(* Schneider Machine Expert - Basic project demo3, file version 2.2.0.0 *)
(* CompanyInformations: WebSite=https://ics-cybersecurity.academy *)
(* ProjectInformations: Name=ICSJWG demo 3 and +, Description=Demonstrate how to program the PLC so that the SCADA can collect some interesting data for cybersecurity *)
(* UserInformations: LastName=Arnaud, FirstName=SOULLIE, Email=asoullie@ics-cybersecurity.academy *)

HARDWARE
  Cpu 0: TM221ME16R/G
  EthernetConfiguration: NetworkName=M221, IpAllocationMode=FixedAddress, IpAddress=192.168.0.53, SubnetMask=255.255.255.0
  SerialLineConfiguration: Baud=Baud19200, Parity=ParityEven, DataBits=DataBits8, StopBits=StopBits1, PhysicalMedium=PhysicalMediumRs485, TransmissionMode=TransmissionModeModbusRtu, SlaveId=1, Addressing=SlaveAddressing
  MastTask: UsePeriodScanMode=false, PeriodScan=100
  FastTask: Period=255
  CpuBehavior: StartingMode=StartAsPreviousState, AutoSaveRamOnEeprom=true, WatchdogPeriod=250

SYMBOLS  (address, symbol, comment, settings)
  %M0       TIMER_START
  %M20      WASH_INTAKE
  %M23      BARREL_VALVE
  %M100     IO_FORCED
  %M101     INPUT_FORCED
  %M102     OUTPUT_FORCED
  %S12      SB_RUNMODE  "The controller is running"
  %S14      SB_IOFORCED  "This bit indicates there is at least one input or output forced"
  %S15      SB_INFORCED  "This bit indicates there is at least one input forced"
  %S16      SB_OUTFORCED  "This bit indicates there is at least one output forced"
  %SW6      SW_CONTROLSTATUS  "Controller Status: NO CONFIG (0), STOP (2), RUN (3), HALT (4), POWERLESS MODE (5)"
  %SW7      SW_STATE  "This word shows the state of the controller (see online help for details)"
  %SW15     SW_FW1VERSION  "Contains the Firmware version of the controller (1st word)"
  %SW16     SW_FW2VERSION  "Contains the Firmware version of the controller (2nd word)"
  %SW30     SW_LASTSCAN1  "Shows execution time of the last controller scan cycle (in ms).If the scan time is 2,250 ms, %SW30 = 2 and %SW70 = 250"
  %SW70     SW_LASTSCAN2  "Shows the microseconds of the execution time of the last controller scan cycle. If the scan time is 2,250 ms the %SW30 will be 2 and the %SW70 = 250"
  %SW94     SW_SIGNATURE  "Contains the signature, changes in case of an application change, in terms of configuration or programming data"
  %MW0      TIMER_DURATION
  %MW10     STILL_TEMP
  %MW11     STILL_LEVEL
  %MW12     CONDENSER_TEMP
  %MW13     BARREL_LEVEL
  %MW21     HEATER
  %MW22     COOLING_PUMP
  %MW100    BOOTLOADER_VERSION
  %MW101    COMMERCIAL_VERSION
  %MW102    FIRMWARE_V_PART1
  %MW103    FIRMWARE_V_PART2
  %MW104    APPLICATION_SIGNATURE
  %MW110    LAST_SCAN_TIME
  %TM0        [Preset=10, Base=OneSecond]

POU Timer
  (* SectionNumber=1 *)

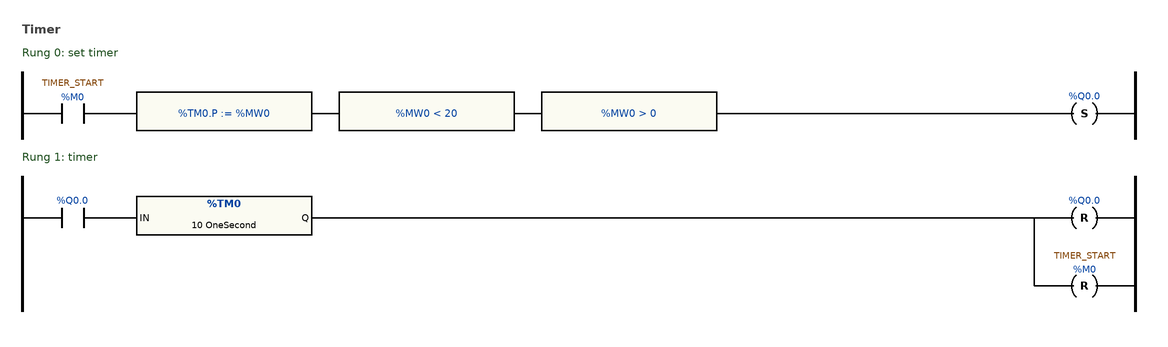

// Rung 0: set timer
  LD %M0                  (* TIMER_START *)
  OPER [ %TM0.P := %MW0 ] (* TIMER_DURATION *)
  AND [ %MW0 < 20 ]       (* TIMER_DURATION *)
  AND [ %MW0 > 0 ]        (* TIMER_DURATION *)
  S %Q0.0
  // as ST:
  //   IF TIMER_START THEN %TM0.P := TIMER_DURATION; END_IF;
  //   IF TIMER_START AND TIMER_DURATION < 20 AND TIMER_DURATION > 0 THEN %Q0.0 := TRUE; END_IF;

// Rung 1: timer
  BLK %TM0
  LD %Q0.0
  IN
  OUT_BLK
  LD Q
  R %Q0.0
  R %M0                   (* TIMER_START *)
  END_BLK
  // as ST:
  //   %TM0(IN := %Q0.0);
  //   IF %TM0.Q THEN %Q0.0 := FALSE; END_IF;
  //   IF %TM0.Q THEN TIMER_START := FALSE; END_IF;

POU Monitoring
  (* SectionNumber=2 *)

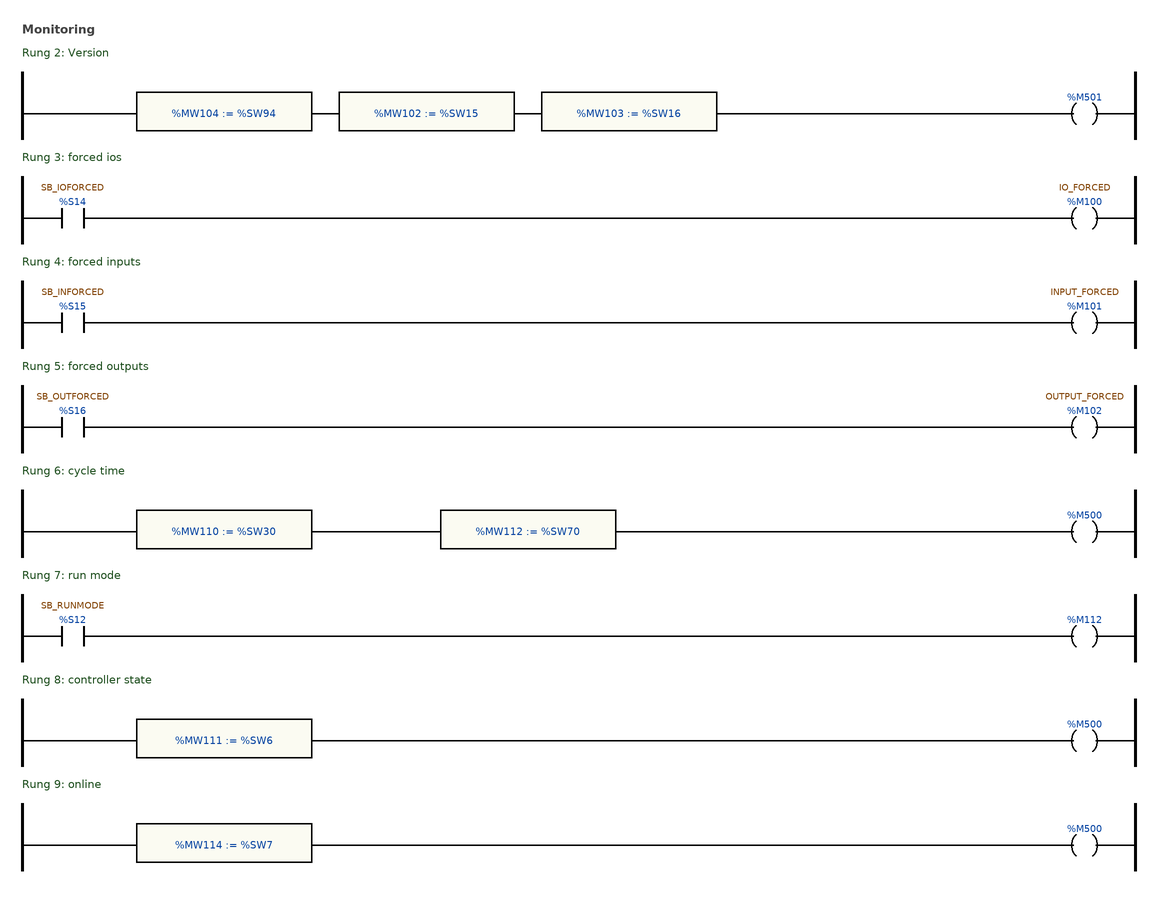

// Rung 2: Version
  LD 1
  OPER [ %MW104 := %SW94 ](* APPLICATION_SIGNATURE, SW_SIGNATURE *)
  OPER [ %MW102 := %SW15 ](* FIRMWARE_V_PART1, SW_FW1VERSION *)
  OPER [ %MW103 := %SW16 ](* FIRMWARE_V_PART2, SW_FW2VERSION *)
  ST %M501
  // as ST:
  //   APPLICATION_SIGNATURE := SW_SIGNATURE;
  //   FIRMWARE_V_PART1 := SW_FW1VERSION;
  //   FIRMWARE_V_PART2 := SW_FW2VERSION;
  //   %M501 := TRUE;

// Rung 3: forced ios
  LD %S14                 (* SB_IOFORCED *)
  ST %M100                (* IO_FORCED *)
  // as ST:
  //   IO_FORCED := SB_IOFORCED;

// Rung 4: forced inputs
  LD %S15                 (* SB_INFORCED *)
  ST %M101                (* INPUT_FORCED *)
  // as ST:
  //   INPUT_FORCED := SB_INFORCED;

// Rung 5: forced outputs
  LD %S16                 (* SB_OUTFORCED *)
  ST %M102                (* OUTPUT_FORCED *)
  // as ST:
  //   OUTPUT_FORCED := SB_OUTFORCED;

// Rung 6: cycle time
  LD 1
  OPER [ %MW110 := %SW30 ](* LAST_SCAN_TIME, SW_LASTSCAN1 *)
  OPER [ %MW112 := %SW70 ](* SW_LASTSCAN2 *)
  ST %M500
  // as ST:
  //   LAST_SCAN_TIME := SW_LASTSCAN1;
  //   %MW112 := SW_LASTSCAN2;
  //   %M500 := TRUE;

// Rung 7: run mode
  LD %S12                 (* SB_RUNMODE *)
  ST %M112
  // as ST:
  //   %M112 := SB_RUNMODE;

// Rung 8: controller state
  LD 1
  OPER [ %MW111 := %SW6 ] (* SW_CONTROLSTATUS *)
  ST %M500
  // as ST:
  //   %MW111 := SW_CONTROLSTATUS;
  //   %M500 := TRUE;

// Rung 9: online
  LD 1
  OPER [ %MW114 := %SW7 ] (* SW_STATE *)
  ST %M500
  // as ST:
  //   %MW114 := SW_STATE;
  //   %M500 := TRUE;
